FUNCTION_BLOCK PAMPlatformscale EXTENDS PAProcessModule
VAR_INPUT
END_VAR
VAR_OUTPUT
END_VAR
VAR
	_PAPointMatIn1 : PAPoint(THIS^);
	_PAPointMatOut1 : PAPoint(THIS^);
END_VAR

METHOD FB_init : BOOL
VAR_INPUT
	bInitRetains : BOOL; // if TRUE, the retain variables are initialized (warm start / cold start)
	bInCopyCode : BOOL;  // if TRUE, the instance afterwards gets moved into the copy code (online change)
	parent : IACComponent;
END_VAR
AddPoint(_PAPointMatIn1);
AddPoint(_PAPointMatOut1);
END_METHOD

PROPERTY PUBLIC PAPointMatIn1 : IACPoint
GET
PAPointMatIn1 := _PAPointMatIn1;
END_GET
END_PROPERTY

PROPERTY PUBLIC PAPointMatOut1 : IACPoint
GET
PAPointMatOut1 := _PAPointMatOut1;
END_GET
END_PROPERTY

END_FUNCTION_BLOCK

(* stored: Version 1.1.0.1, ProductVersion 3.1.4020.12
   POU PAMPlatformscale: Id {9833b039-f9b1-4cf8-89e9-1913eb68accb}, SpecialFunc None
   Method FB_init: Id {42614e4c-ef3f-45fd-a399-8b5b102563d1}
   Property PAPointMatIn1: Id {c537a64e-8d27-4844-9398-00aa172a0bc6}
   Get Get: Id {5bc0117b-b9d2-41a8-850d-990c45b579fa}
   Property PAPointMatOut1: Id {76edb520-db86-47d6-b0a5-7a67dbf6d0c6}
   Get Get: Id {181c9bb3-bac5-4931-b1d1-c0234f51b6ea} *)
